FUNCTION IsEqualAnyType : BOOL
VAR_INPUT
	a					: __SYSTEM.AnyType; // A and B have to be same type
	b					: __SYSTEM.AnyType; // A and B have to be same type
END_VAR

IF a.TypeClass <> b.TypeClass THEN
	RETURN;
END_IF

IsEqualAnyType := MEMCMP(a.pValue, b.pValue, a.diSize) = 0;

END_FUNCTION

(* stored: Version 1.1.0.1, ProductVersion 3.1.4024.12
   POU IsEqualAnyType: Id {306151ac-6fe4-0968-06fe-fd616840ca54}, SpecialFunc None *)
